// TwinCAT 3 PLC project TcUnits
// Title: TcUnits
// Company: Roald
// Author: Roald Ruiter
// ProjectVersion: 0.1.1
// Description: Aliases for units
// ProgramVersion: 3.1.4023.0
// project tree:
//   Acceleration/ MillimeterPerSecondSquared.TcDUT
//   Distance/ Millimeter.TcDUT
//   Force/ Newton.TcDUT (not stored)
//   / Percent.TcDUT
//   Speed/ MillimeterPerSecond.TcDUT (not stored)
//   Time/ Millisecond.TcDUT (not stored)
//   Torque/ NewtonMeter.TcDUT
//   Weight/ Kilogram.TcDUT (not stored)
// real-time tasks:
//   TASK PlcTask: cycle T#10ms, priority 20, ADS port 350

// ---- Acceleration/MillimeterPerSecondSquared.TcDUT
TYPE MillimeterPerSecondSquared : LREAL;
END_TYPE

// ---- Distance/Millimeter.TcDUT
TYPE Millimeter : LREAL;
END_TYPE

// ---- Percent.TcDUT
TYPE Percent : LREAL;
END_TYPE

// ---- Torque/NewtonMeter.TcDUT
TYPE NewtonMeter : LREAL;
END_TYPE
